Staubli VAL3: getDistance.pgx

public program getDistance(tool x_tTool (dimensions=1), num& x_nDistance[] (dimensions=1), bool x_bCycle (dimensions=1), num x_nIndex (dimensions=1))
  local num l_nValue
  local point l_pActual
  local point l_pPoint
  local point l_pPrev
  local trsf l_trsfEmpty
begin
  // first point
  if x_nIndex==0
    x_nDistance=10
    return
  else
    //
    // get the point
    //
    call getPoint(l_pActual,x_bCycle,x_nIndex)
    call getPoint(l_pPrev,x_bCycle,x_nIndex-1)
    if x_bCycle
      x_nDistance=distance(l_pPrev.trsf,l_trsfEmpty)
    else
      x_nDistance=distance(l_pPrev.trsf,l_trsfEmpty)
    endIf
  endIf
end
